(* CoDeSys 2.3 export: Struct.ftl *)

(* Data type in <#if path?has_content><#list path as dir>/${dir}</#list></#if> *)
TYPE ${name} :
STRUCT
<#if vars?has_content>
<#list vars as var>
    ${var.name}: ${var.type}<#if var.value??> := ${var.value}</#if>;
</#list>
</#if>
END_STRUCT
END_TYPE
